// TIA Portal V16 program export: 0 tag tables, 0 data types, 0 data blocks, 2 code blocks (in call order from the OBs), 0 instance data blocks

ORGANIZATION_BLOCK "Main"   // OB1, LAD, ProgramCycle
TITLE = "Main Program Sweep (Cycle)"
{ S7_Optimized_Access := 'TRUE' }
VERSION : 0.1
// stored: AutoNumber true, IsIECCheckEnabled false, SetENOAutomatically false
BEGIN

REGION Network 1
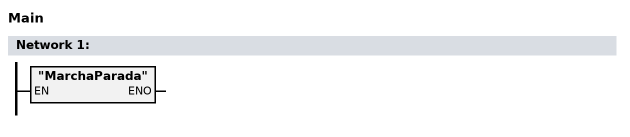
   RUNG wire#powerrail
      "MarchaParada"()
   END_RUNG
   // the same network as SCL:
   "MarchaParada"();
END_REGION
END_ORGANIZATION_BLOCK

FUNCTION "MarchaParada" : Void   // FC1, LAD
{ S7_Optimized_Access := 'TRUE' }
VERSION : 0.1
// stored: AutoNumber true, IsIECCheckEnabled false, SetENOAutomatically false, UDAEnableTagReadback false
BEGIN

REGION Network 1
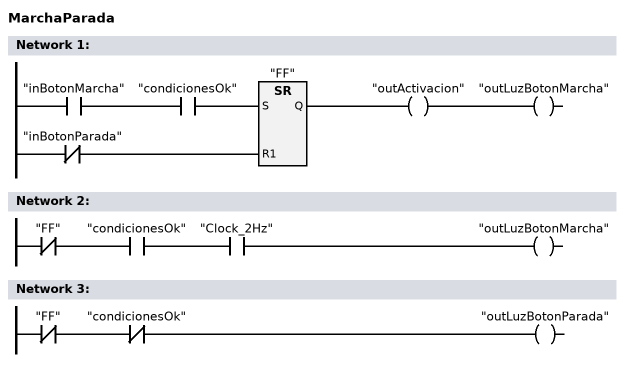
   RUNG wire#powerrail
      Contact( "inBotonMarcha" )
      Contact( "condicionesOk" )
      S_SR(operand := "FF", r1 := wire#w1)
      Coil( "outActivacion" )
      Coil( "outLuzBotonMarcha" )
   END_RUNG
   RUNG wire#powerrail
      I_Contact( "inBotonParada" )
   END_RUNG wire#w1
   // the same network as SCL:
   IF "inBotonMarcha" AND "condicionesOk" THEN
       "FF" := TRUE;   // SR flip-flop
   END_IF;
   IF NOT "inBotonParada" THEN "FF" := FALSE; END_IF;
   "outActivacion" := "FF";
   "outLuzBotonMarcha" := "FF";
END_REGION

REGION Network 2
   RUNG wire#powerrail
      I_Contact( "FF" )
      Contact( "condicionesOk" )
      Contact( "Clock_2Hz" )
      Coil( "outLuzBotonMarcha" )
   END_RUNG
   // the same network as SCL:
   "outLuzBotonMarcha" := NOT "FF" AND "condicionesOk" AND "Clock_2Hz";
END_REGION

REGION Network 3
   RUNG wire#powerrail
      I_Contact( "FF" )
      I_Contact( "condicionesOk" )
      Coil( "outLuzBotonParada" )
   END_RUNG
   // the same network as SCL:
   "outLuzBotonParada" := NOT "FF" AND NOT "condicionesOk";
END_REGION
END_FUNCTION
